# EPICS IOC start-up script: iocsh/ethercatmcShutter.iocsh
ethercatmcCreateIndexerAxis("$(MOTOR_PORT)", "$(AXIS_NO)", "6", "$(AXISCONFIG)")

ethercatmcCreateAsynParam $(MOTOR_PORT) AUXBITOpened Int32
ethercatmcCreateAsynParam $(MOTOR_PORT) AUXBITClosed Int32

dbLoadRecords("ethercatmcShutter.template", "PREFIX=$(PREFIX), R=$(R), DESC=$(DESC), MOTOR_PORT=$(MOTOR_PORT), AXIS_NO=$(AXIS_NO)")
